FUNCTION_BLOCK Ex70x7_DMC_Channel
VAR_INPUT
END_VAR
VAR_OUTPUT
END_VAR
VAR
	ENCStatus AT%I* : StepperENCStatus;
	STMStatus AT%I* : StepperSTMStatus;
	POSStatus AT%I* : StepperPOSStatus;
	
	ENCControl AT%Q* : StepperENCControl;
	STMControl AT%Q* : StepperSTMControl;
	POSControl AT%Q* : StepperPOSControl;
	
	_InTarget : BOOL;
	
	State :(
		_00_mWait,
        _01_mReset,
        _02_mEnable,
		_06_mGotoPosition,
		_07_mStop,
		_08_mSetPosition,
		_09_RunAtExternalVelo,
		_10_Disable);
		
	tonHoldHigh				: ton;
END_VAR

CASE State OF
        _00_mWait : 
			;
        _01_mReset : 
			STMControl.Reset := TRUE;
			tonHoldHigh(in := TRUE, pt := T#500MS);
			IF tonHoldHigh.Q THEN
				STMControl.Reset := FALSE;
				IF STMStatus.Error = FALSE AND
					STMStatus.Warning = FALSE AND
					STMStatus.Ready = TRUE
				THEN
					State := _00_mWait;
					tonHoldHigh(in := FALSE, pt := T#500MS);
				END_IF
			END_IF
			
        _02_mEnable : 
			IF STMStatus.Error THEN				
				State := _01_mReset;
			ELSE
				STMControl.Enable := TRUE;			
			END_IF
			
		_06_mGotoPosition :
			POSControl.Execute := TRUE;
			_InTarget := FALSE;
			IF POSStatus.InTarget THEN
				State := _02_mEnable;
				POSControl.Execute := FALSE;
				_InTarget := TRUE;
			END_IF
			
		_07_mStop : 
			POSControl.Execute := FALSE;
			IF POSStatus.ReadyToExecute THEN	
				State := _02_mEnable;
			END_IF
			
		_08_mSetPosition :
			POSControl.Execute := TRUE;
			
			IF POSStatus.Calibrated THEN
				POSControl.Execute := FALSE;
				State := _02_mEnable;
			END_IF
			
		_09_RunAtExternalVelo :
			POSControl.Execute := TRUE;
			_InTarget := false;
			
		_10_Disable:
			STMControl.Enable := FALSE;
			State := _00_mWait;
		
			
END_CASE

PROPERTY ActualPosition : lreal
GET
ActualPosition := UDINT_TO_LREAL( POSStatus.ActualPosition)/8062.72;
END_GET
END_PROPERTY

PROPERTY ActualVelocity : int
GET
ActualVelocity := POSStatus.ActualVelocity;
END_GET
END_PROPERTY

METHOD CalibrateMotor : BOOL
VAR_INPUT
END_VAR
IF State = _02_mEnable THEN
	State := _08_mSetPosition;
	//POSControl.Velocity := REAL_TO_INT( Velocity*252);
	POSControl.StartType := StartType.Calibrate;
	//POSControl.TargetPosition := LREAL_TO_UDINT(Position*8062.72);
	//POSControl.TargetPosition := LREAL_TO_UDINT(Position*10);
END_IF
END_METHOD

METHOD Disable : BOOL
VAR_INPUT
END_VAR
IF STMStatus.Ready THEN
	State := _10_Disable;
END_IF
END_METHOD

METHOD Enable : BOOL
VAR_INPUT
END_VAR
IF STMStatus.ReadyToEnable THEN
	State := _02_mEnable;
END_IF
END_METHOD

METHOD GoToPosition : BOOL
VAR_INPUT
	Position : LREAL;
	Velocity : REAL;
END_VAR
IF State = _02_mEnable THEN
	State := _06_mGoToPosition;
	POSControl.Velocity := REAL_TO_INT( Velocity*252);
	POSControl.StartType := StartType.Absolute;
	POSControl.TargetPosition := LREAL_TO_UDINT(Position*8062.72);
END_IF
END_METHOD

PROPERTY InTarget : bool
GET
InTarget := _InTarget;
END_GET
END_PROPERTY

METHOD MoveAtVelocity : BOOL
VAR_INPUT
	Velocity : REAL;
END_VAR
IF State = _02_mEnable THEN
	State := _09_RunAtExternalVelo;
	POSControl.Velocity := REAL_TO_INT( Velocity*252);
	POSControl.StartType := StartType.VeloPositive;
END_IF
END_METHOD

PROPERTY Ready : bool
GET
Ready := STMStatus.Ready;
END_GET
END_PROPERTY

METHOD Reset : BOOL
VAR_INPUT
END_VAR
IF STMStatus.Error OR STMStatus.Warning OR POSStatus.Error THEN
	State := _01_mReset;
END_IF
END_METHOD

METHOD Stop : BOOL
VAR_INPUT
END_VAR
IF POSControl.Execute THEN
	State  := _07_mStop;
END_IF
END_METHOD

END_FUNCTION_BLOCK

(* stored: Version 1.1.0.1, ProductVersion 3.1.4024.11
   POU Ex70x7_DMC_Channel: Id {165026ab-25d1-406b-8c2e-dceb74646d34}, SpecialFunc None
   Property ActualPosition: Id {87402dda-3934-4e72-a117-2fd73b8f7cfc}
   Get Get: Id {9e3576a2-691e-4a64-8b2c-f8318dfb70e0}
   Property ActualVelocity: Id {e6b14254-e519-45f2-8f01-a31ccc3b9831}
   Get Get: Id {87355008-d361-4495-a8e1-ec6ab95b56e2}
   Method CalibrateMotor: Id {66ad0482-651d-4769-959d-9a03b9363113}
   Method Disable: Id {b3eb0936-8c9c-40c1-98cc-33098a295206}
   Method Enable: Id {1a8f71be-b4c5-43c0-8b97-fbf99520c81a}
   Method GoToPosition: Id {e811e2fb-700f-45d5-986c-8b7c09a4b4bd}
   Property InTarget: Id {45d1a00c-f015-4275-9637-dcc7fb103714}
   Get Get: Id {348b89ca-9997-4f57-90d2-2af53e069e66}
   Method MoveAtVelocity: Id {a3e3882f-4f97-4cee-9501-79a6538b7718}
   Property Ready: Id {49e3df1c-7e75-46cd-8d98-5c00c69b033e}
   Get Get: Id {2d0fadb1-ac1c-40d3-833e-2a14060a65a0}
   Method Reset: Id {642776ce-ed1f-4014-bd07-da23a37a2d66}
   Method Stop: Id {e6eed7a9-3f7b-4998-9d25-a5f6272d282c} *)
